FUNCTION_BLOCK FB_Count
VAR_INPUT
	bInput				:	BOOL;	
	bAllFlanks			:	BOOL := FALSE;				//Alle Flanken verwenden?
	rMultiplier			:	REAL := 1;					//Wert wirt mit wOut multipliziert
	iFactor				:	INT	:= 1;					//Factor to shift komma
END_VAR
VAR_OUTPUT
	wOut				:	WORD;
END_VAR
VAR_IN_OUT
	wCountRetain		:	WORD;
END_VAR
VAR
	fbRTrig				:	R_TRIG;
	fbFTrig				:	F_TRIG;
	
	iMaxValue			:	UINT := 65535;
END_VAR


fbRTrig(CLK:= bInput, Q=> );

IF fbRTrig.Q THEN
	wCountRetain := TO_WORD((wCountRetain + 1) MOD iMaxValue);
END_IF	

IF bAllFlanks THEN
	fbFTrig(CLK:= bInput, Q=> );

	IF fbFTrig.Q THEN
		wCountRetain := TO_WORD((wCountRetain + 1) MOD iMaxValue);
	END_IF	
END_IF
	
wOut	:= REAL_TO_WORD((wCountRetain * rMultiplier)*iFactor);

END_FUNCTION_BLOCK

(* stored: Version 1.1.0.1, ProductVersion 3.1.4024.13
   POU FB_Count: Id {7eccf564-e373-4dac-ab77-0db3104eaba8}, SpecialFunc None *)
